// TIA Portal V18 export
TYPE "LGasp_TypeCoil_fromERP"
// stored: IsFailsafeCompliant false
   STRUCT
      CoilCode : WString[30];   // Codice alfanumerico identificatico del coil
      MaterialType : WString[30];   // Tpo di materiale
      Width : LReal;   // [mm]
      Thickness : LReal;   // [mm]
      Weight : LReal;   // [kg]
   END_STRUCT;
END_TYPE
